FUNCTION CalcBreakTime : TIME
VAR_INPUT
    iWorkSessions : INT;   (* number of finished work blocks *)
END_VAR

(* Long break after every 4th work block, short break otherwise *)
IF (iWorkSessions > 0) AND ((iWorkSessions MOD 4) = 0) THEN
    CalcBreakTime := T#15m;    (* long break *)
ELSE
    CalcBreakTime := T#5m;     (* short break *)
END_IF

END_FUNCTION

(* stored: Version 1.1.0.1, ProductVersion 3.1.4024.16
   POU CalcBreakTime: Id {f84bf3ae-d4e2-4b8e-b080-cad5e50516b3}, SpecialFunc None *)
